TYPE SensorBeckhoffIO_In :
	STRUCT
		ValuesRaw 		: INT;
	END_STRUCT
END_TYPE

(* stored: Version 1.1.0.1
   DUT SensorBeckhoffIO_In: Id {31721cda-486d-0974-3faa-63c5e18a66e6} *)
